# EPICS autosave request: utcaApp/Db/ebpm_ioc.req
file "bpm_common.req", P=${P}, R=${R}, P1=${P1}, R1=${R1}, P2=${P2}, R2=${R2}

file "ebpm_single.req", P=${P1}, R=${R1}
file "ebpm_single.req", P=${P2}, R=${R2}
